FUNCTION_BLOCK StationBehaviour IMPLEMENTS I_Cyclic, I_Resettable, I_Object
VAR
	State : StationBehaviourState;  
	CurrentStation : UINT;
	TargetStationPosition : MC_LREAL;
	_MoverVelocity : MC_LREAL := 1000.0;
	stSequenceInfo : StationBehaviourInfo;
	StationNumber : INT;
	StationArray : ARRAY[0..19] OF I_Station;
	Process : IProcess;
	ThisMover : I_XtsMover;
	ExecuteSequence : BOOL;
	_startPosition : MC_LREAL;
	_XtsNoHome : BOOL;
	_NonModuloMoves : BOOL := FALSE;
END_VAR

{analysis -2}

PROPERTY AbsoluteMoves : bool
GET
AbsoluteMoves := _NonModuloMoves;
END_GET
SET
_NonModuloMoves := AbsoluteMoves;
END_SET
END_PROPERTY

METHOD PUBLIC Cycle : HRESULT
VAR_INPUT
END_VAR
CASE State OF
	StationBehaviourState.WaitForMoverEnabled:
		IF ThisMover.IsEnabled THEN
			State := StationBehaviourState.WaitingForStart;
		END_IF
		
	StationBehaviourState.WaitingForStart:
		IF ExecuteSequence THEN
			State := StationBehaviourState.MovingToStart;
		END_IF
		
	StationBehaviourState.MovingToStart:
		IF ThisMover.isMoverAtPosition(position := _startPosition) OR _XtsNoHome THEN
			State := StationBehaviourState.MoveToFirstStation;
		END_IF
			
	StationBehaviourState.MoveToFirstStation:
		IF StationArray[CurrentStation] <> 0 THEN
			IF SUCCEEDED(ThisMover.MoveTo(RequiredPosition := StationArray[CurrentStation].Position,
								MoveVelocity := _MoverVelocity,
								NonModuloMove := _NonModuloMoves)) THEN
								
				TargetStationPosition := StationArray[CurrentStation].Position;
				State := StationBehaviourState.MovingToCurrentStation;
			END_IF
		END_IF

	StationBehaviourState.MovingToCurrentStation:
		IF ThisMover.IsStationary THEN 
			IF ThisMover.isMoverAtPosition(TargetStationPosition) THEN
				State := StationBehaviourState.ArrivedAtStation;
			ELSE
				State := StationBehaviourState.MoverQueueingAtStation;
			END_IF
		END_IF
	
	StationBehaviourState.ArrivedAtStation:
		IF SUCCEEDED(StationArray[CurrentStation].MyMover(ThisMover)) THEN
			IF __QUERYINTERFACE(StationArray[CurrentStation],Process) THEN
				State := StationBehaviourState.StartingProcess;
			ELSE
				State := StationBehaviourState.WaitingForStationComplete;
			END_IF
		END_IF
		
	StationBehaviourState.MoverQueueingAtStation:
		IF NOT ThisMover.IsStationary THEN
				State := StationBehaviourState.MovingToCurrentStation;
		END_IF

	StationBehaviourState.WaitingForStationComplete:
		IF StationArray[CurrentStation].isComplete() THEN
			State := StationBehaviourState.CheckIfFinalStation;
		END_IF

	StationBehaviourState.StartingProcess:
		ThisMover.MoveTo(RequiredPosition := Process.EndPosition,
								MoveVelocity := Process.ProcessVelocity,
								NonModuloMove := _NonModuloMoves);
		State := StationBehaviourState.MoverInProcess;
								
	StationBehaviourState.MoverInProcess:
		IF ThisMover.IsStationary THEN 
			IF ThisMover.isMoverAtPosition(Process.EndPosition) THEN
				State := StationBehaviourState.CheckIfFinalStation;
			END_IF
		END_IF
	
	StationBehaviourState.CheckIfFinalStation:
		IF CurrentStation = StationNumber - 1 THEN
			CurrentStation := 0; 
			TargetStationPosition := StationArray[CurrentStation].Position;
			IF SUCCEEDED(ThisMover.MoveTo(RequiredPosition := TargetStationPosition,
							MoveVelocity := _MoverVelocity,
							NonModuloMove := _NonModuloMoves)) THEN
				State := StationBehaviourState.MovingToCurrentStation;
			END_IF
		ELSE
			State := StationBehaviourState.MovingToNextStation;
		END_IF
		
	StationBehaviourState.MovingToNextStation:
		TargetStationPosition := StationArray[CurrentStation + 1].Position;
		IF 	SUCCEEDED(ThisMover.MoveTo(RequiredPosition := TargetStationPosition,
							MoveVelocity := _MoverVelocity,
							NonModuloMove := _NonModuloMoves)) THEN	
			CurrentStation := CurrentStation + 1;
			State := StationBehaviourState.MovingToCurrentStation;
		END_IF	
	StationBehaviourState.Stopped;
		IF ExecuteSequence THEN
			TargetStationPosition := StationArray[CurrentStation].Position;
			IF CurrentStation = 0 THEN
				IF 	SUCCEEDED(ThisMover.MoveTo(RequiredPosition := TargetStationPosition,
									MoveVelocity := _MoverVelocity,
									NonModuloMove := _NonModuloMoves)) THEN	
					State := StationBehaviourState.MovingToCurrentStation;
				END_IF	
			ELSE
				IF 	SUCCEEDED(ThisMover.MoveTo(RequiredPosition := TargetStationPosition,
									MoveVelocity := _MoverVelocity,
									NonModuloMove := _NonModuloMoves)) THEN	
					State := StationBehaviourState.MovingToCurrentStation;
				END_IF	
			END_IF
		END_IF
		
	StationBehaviourState.SequenceError:

	ELSE
		Cycle := E_FAIL;
END_CASE

//Cyclic update info data
stSequenceInfo.CurrentStation := UINT_TO_INT(CurrentStation);
stSequenceInfo.MoverId := ThisMover.AxisRef.NcToPlc.AxisId;
stSequenceInfo.State := State;
stSequenceInfo.Velocity := ThisMover.AxisRef.NcToPlc.ActVelo;
END_METHOD

PROPERTY MoverVelocity : mc_lreal
GET
MoverVelocity := _MoverVelocity;
END_GET
SET
_MoverVelocity := MoverVelocity;
END_SET
END_PROPERTY

PROPERTY MyMover : I_XtsMover
GET
MyMover := ThisMover;
END_GET
SET
ThisMover := MyMover;
END_SET
END_PROPERTY

PROPERTY MyStartPosition : MC_LREAL
GET
MyStartPosition := _startPosition;
END_GET
SET
_startPosition := MyStartPosition;
END_SET
END_PROPERTY

METHOD RegisterAStation : HRESULT
VAR_INPUT
	Station : I_Station;
END_VAR
IF Station = 0 THEN
	RegisterAStation  := -1;
	RETURN;
END_IF
StationArray[StationNumber] := Station;
StationNumber := StationNumber + 1;
END_METHOD

METHOD RegisterWithParent
VAR_INPUT
	Parent	: I_HostObjects;
END_VAR
Parent.RegisterCyclic(THIS^);
END_METHOD

METHOD Reset : HRESULT
VAR_INPUT
END_VAR
State := StationBehaviourState.WaitingForStart;
CurrentStation := 0;
TargetStationPosition := 0.0;
stSequenceInfo.CurrentStation := UINT_TO_INT(CurrentStation);
stSequenceInfo.MoverId := ThisMover.AxisRef.NcToPlc.AxisId;
stSequenceInfo.State := State;
stSequenceInfo.Velocity := ThisMover.AxisRef.NcToPlc.ActVelo;
ExecuteSequence := FALSE;
Reset := 1;
END_METHOD

METHOD StartIndexing : BOOL
VAR_INPUT
END_VAR
ExecuteSequence := TRUE;
END_METHOD

METHOD StopIndexing : BOOL
VAR_INPUT
END_VAR
State := StationBehaviourState.Stopped;
ThisMover.HaltAxis();
END_METHOD

PROPERTY XtsNoHome : BOOL
GET
XtsNoHome := _XtsNoHome;
END_GET
SET
_XtsNoHome := XtsNoHome;
END_SET
END_PROPERTY

END_FUNCTION_BLOCK

(* stored: Version 1.1.0.1
   POU StationBehaviour: Id {50af290e-a0d7-45b3-a647-c8828b096bd1}, SpecialFunc None
   Property AbsoluteMoves: Id {17b68adf-bca0-4be6-993f-8e20810fcd58}
   Get Get: Id {9984e65c-22d5-4260-98b6-c2626c7cc30d}
   Set Set: Id {2d9b4a71-c7c5-4acd-9b62-753da375193c}
   Method Cycle: Id {0bc270b2-0e7a-4545-b872-87f2d15ca3f5}
   Property MoverVelocity: Id {4f2224ad-0534-4bd9-a8e4-5b63b7e53b5c}
   Get Get: Id {0bf3cfa6-cc44-4232-989f-70bced017a55}
   Set Set: Id {a9bdfb5a-ef56-4b9e-9f78-288684e24d6c}
   Property MyMover: Id {d0dbd650-93c6-4e7f-a733-abc40a2f12bf}
   Get Get: Id {52e46adf-1b9f-404f-a8d7-de686d91d4ef}
   Set Set: Id {a9693a81-065c-4ba2-8a99-3606c71cf06a}
   Property MyStartPosition: Id {30ed087d-d896-49f8-aaff-c511c0d55a71}
   Get Get: Id {ebcb0d89-302c-4f5d-86e5-f5e15f136ea5}
   Set Set: Id {57b76837-f6ca-44d6-8033-7a2d9ee3e944}
   Method RegisterAStation: Id {14d9a1a8-6162-46e7-9803-61945cdf77e8}
   Method RegisterWithParent: Id {4ad7e011-f71b-4cbe-b657-57f840858ed2}
   Method Reset: Id {01dd3306-e903-4754-85c4-ea13c41e0b8c}
   Method StartIndexing: Id {6e4b7f28-1f53-404c-b56b-f1310c888415}
   Method StopIndexing: Id {6fcff83f-b689-4f39-8c14-494c41dd48fe}
   Property XtsNoHome: Id {7aad9af3-71dc-4b8d-9a2b-19016c2a644b}
   Get Get: Id {d3413585-01ef-4909-a612-e4cda3a7b8e0}
   Set Set: Id {ca6f67d3-9265-4c0f-849c-5e4c98f82e9b} *)
